// TIA Portal V19 export
FUNCTION "PB_Lamp" : Bool   // FC48, LAD
TITLE = PUSH BUTTON LAMP CONTROL
// stored: Access Published, SetENOAutomatically false
   VAR_INPUT
      OpSelect : Bool;
      OpRequest : Bool;
      OpRunning : Bool;
      OpDone : Bool;
   END_VAR
BEGIN

REGION Network 1: Lamp
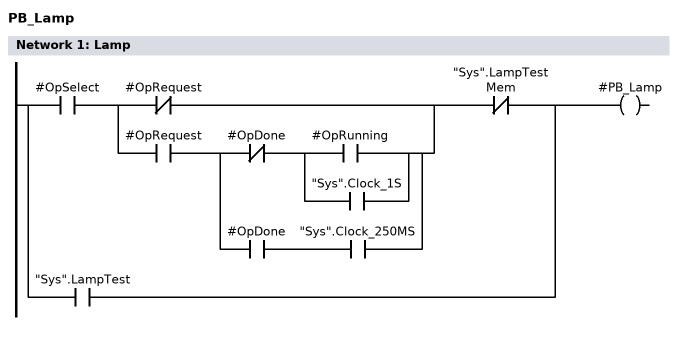
   RUNG wire#powerrail
      Contact( #OpSelect )
      wire#w1
      I_Contact( #OpRequest )
      wire#w2
      I_Contact( "Sys".LampTestMem )
      wire#w5
      Coil( #PB_Lamp )
   END_RUNG
   RUNG wire#w1
      Contact( #OpRequest )
      wire#w3
      I_Contact( #OpDone )
      wire#w4
      Contact( #OpRunning )
   END_RUNG wire#w2
   RUNG wire#w4
      Contact( "Sys".Clock_1S )
   END_RUNG wire#w2
   RUNG wire#w3
      Contact( #OpDone )
      Contact( "Sys".Clock_250MS )
   END_RUNG wire#w2
   RUNG wire#powerrail
      Contact( "Sys".LampTest )
   END_RUNG wire#w5
   // the same network as SCL:
   #PB_Lamp := (#OpSelect AND (NOT #OpRequest OR (#OpRequest AND ((NOT #OpDone AND (#OpRunning OR "Sys".Clock_1S)) OR (#OpDone AND "Sys".Clock_250MS)))) AND NOT "Sys".LampTestMem) OR "Sys".LampTest;
END_REGION
END_FUNCTION
